{attribute 'qualified_only'}
{attribute 'strict'}
TYPE cTraySize :
(
	
	NoSize := 0,
	Small:= 1,
	Large := 2
	
) DINT;
END_TYPE

(* stored: Version 1.1.0.1, ProductVersion 3.1.4024.6
   DUT cTraySize: Id {20470f2b-2a39-423b-8833-f0729c11e101} *)
